// TwinCAT 3 PLC project Testbench
// Title: Testbench
// Company: Zeugwerk GmbH
// Author: Zeugwerk GmbH
// ProjectVersion: 1.7.2.1
// Description: Lightweight unit-test (adapter) library to be used together with Zeugwerk Creator (Test Explorer)
// ProgramVersion: 3.1.4023.0
// project tree:
//   / IAssertions.TcIO (not stored), ITestContext.TcIO, IUnitTest.TcIO

// ---- ITestContext.TcIO
/// A context can be passed to every unittest in order to implement tests, which take several cycles of the PLC to complete.
/// Also, for a test suite the context is retained, and [UserData](xref:ZCore.ITestContext#UserData) can be used to pass
/// data between tests if needed.
///
/// When implementing tests with a context, the signature of the tests have to look like
/// ``` st  
/// METHOD Test_<NAME OF THE TEST>
/// VAR_INPUT
///   context : ITestContext;
/// END_VAR
/// ```
///
/// The `context` provides properties to control the flow of the tests and `context.Assertions` can be used to 
/// implement checks in the test.
INTERFACE ITestContext

/// Returns the assertion interface, which can be used to do checks in a test case.
PROPERTY Assertions : IAssertions
GET
END_GET
END_PROPERTY

/// When set to `TRUE` the unit tests will be continously called until `Busy=FALSE`. This is useful
/// if a test case has a time dependency, which can not simply be mocked. 
PROPERTY Busy : BOOL
GET
END_GET
SET
END_SET
END_PROPERTY

/// UserData can be set and retrieved from a context to pass along information between different test cases.
/// To use it, create your own datastructure and pass a pointer to `UserData`
///
/// For instance, you can create a datastructure, which looks like
/// ``` st 
/// TYPE MyTestData :
/// STRUCT
///   MyTestVar : INT;
/// END_STRUCT
/// ```
///
/// Then in a test case, set an instance of the structure to the context (note the instance has to be created on the heap, e.g. VAR_INST).
PROPERTY UserData : POINTER TO BYTE
GET
END_GET
SET
END_SET
END_PROPERTY

END_INTERFACE

// ---- IUnitTest.TcIO
/// Unittests are handled by Zeugwerk Developer-Tools, which are paritially available as online services in the form of
/// GitHub actions ([zkbuild](https://github.com/Zeugwerk/zkbuild-action), [zkdoc](https://github.com/Zeugwerk/zkdoc-action).
/// These online services are available for any PLC and do not explicitly require the Zeugwerk Framework, as demonstrated by
/// open source projects
/// - [Twinson](https://github.com/stefanbesler/Twinson)
/// - [Struckig](https://github.com/stefanbesler/struckig)
///
/// The unittest mechanism is as follows
/// 1. Testsuites are implemented as function blocks, which have to implement [IUnitTest](xref:Testbench.IUnitTest)
///
///    ``` st  
///    FUNCTION_BLOCK <POU>Test EXTENDS <POU> IMPLEMENTS Testbench.IUnitTest>
///    ```
///   
///    Note that by extending testsuites from the object that is testes, the suite gets access protected methods
///    of the POU.
/// 1. Tests are implemented as method for each testsuite. Methods, which are considered unittests follow the following signature.
///
///    ``` st  
///    METHOD Test_<NAME OF THE TEST>
///    VAR_INPUT
///      assertions : IAssertions;
///    END_VAR
///    ```
///
///    or, for more simple tests with only 1 assertion
///
///    ``` st  
///    METHOD Test_<NAME OF THE TEST>
///    VAR_OUTPUT
///      expected : <TYPE>;
///      actual : <TYPE>;
///      message : STRING(255);
///    END_VAR
///    ```
///    where `<TYPE>` can be any IEC61131-3 compatible type like DINT, INT, WORD or BOOL
/// 1. Test may be parametrized by using the `DataRow` attribute. When generating the unittest, every datarow will be its own test. The signature
///    for using paramtrized tests looks as follows.
///
///    ``` st  
///    {attribute 'DataRow(<PARAMETER_1 VALUE>, <PARAMETER_2 VALUE>, ..., <PARAMETER_N VALUE>)'}
///    {attribute 'DataRow(<PARAMETER_1 VALUE>, <PARAMETER_2 VALUE>, ..., <PARAMETER_N VALUE>)'}
///    // ...
///    {attribute 'DataRow(<PARAMETER_1 VALUE>, <PARAMETER_2 VALUE>, ..., <PARAMETER_N VALUE>)'}
///    METHOD Test_<NAME OF THE TEST>
///    VAR_INPUT
///      assertions : IAssertions;
///      <PARAMETER_1> : <PARAMETER_1 DATATYPE>
///      <PARAMETER_2> : <PARAMETER_2 DATATYPE>
///      // ...
///      <PARAMETER_N> : <PARAMETER_N DATATYPE>
///    END_VAR
///    ```
INTERFACE IUnitTest

END_INTERFACE
